RoboDK station: New Station (2).rdk

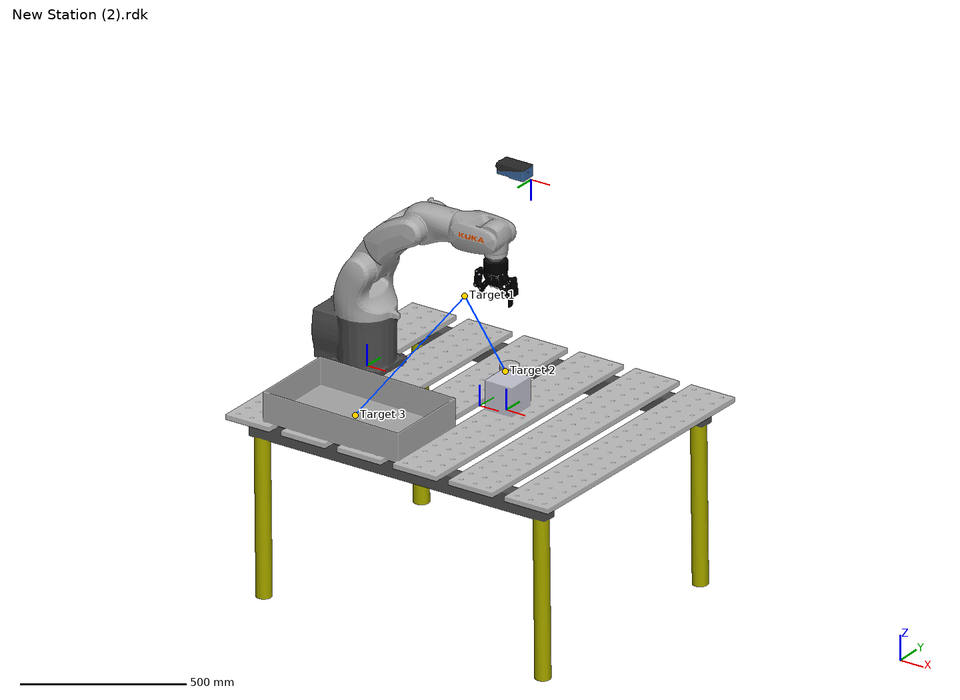
[picture v0: the station drawn from its stored meshes, robots at their saved joint values, targets as dots, program paths as lines]
Station New Station (2). Poses are relative to the parent item; angles as X-Y-Z fixed-axis rotations.
Station parameters (name, value as stored): IO_5, 1, CollisionFreePlanner, KUKA KR 3 R540, CollisionFreePlanner-Rob KUKA KR 3 R540
  - frame KUKA KR 3 R540 Base at (-517.33, 1.06, 0.26) mm, rotated rx -0.44 ry -1.04 rz -0.63 deg
    - robot KUKA KR 3 R540: 6 axes, payload 3 kg, reach 541 mm, repeatability 0.02 mm, weight 26 kg
        modified DH rows (alpha deg, a mm, theta deg, d mm): 0, 0, 0, 345; -90, 20, 0, 0; 0, 260, -90, 0; -90, 20, 0, 260; 90, 0, 0, 0; -90, 0, 180, 75
        joint limits [-170, -170, -110, -175, -120, -350] to [170, 50, 155, 175, 120, 350]; home [0, -90, 90, 0, 0, 0]; saved at [-2.236, -43.368, 43.433, -0.46, 90.207, -1.607]
      - tool Gripper RobotiQ 85 Opened, TCP at (0, -20, 130) mm, size 147.4 x 146.8 x 75 mm
      - tool Gripper RobotiQ 85 Closed, TCP at (0, -20, 130) mm, size 134.4 x 157.6 x 75 mm
    - frame Frame 2 at (440.16, -30.43, -6.02) mm
      - target Target 1 (Cartesian target) at (-55.66, 5.41, 346.75) mm, rotated rx -180 ry 0.75 rz 180 deg; joints [0.676, -64.85, 76.675, 0.003, 78.427, 0.675] of KUKA KR 3 R540
      - target Target 2 (Cartesian target) at (6.97, 122.8, 68.55) mm, rotated rx 180 ry 0.75 rz -180 deg; joints [-14.168, -20.802, 65.869, -0.087, 45.177, -14.106] of KUKA KR 3 R540
      - target Target 3 (Cartesian target) at (-168.25, -408.46, 82.33) mm, rotated rx -180 ry 0.75 rz 180 deg; joints [56.988, -14.801, 48.393, 0.254, 56.546, 56.848] of KUKA KR 3 R540
      - object Table at (0, 0, 0) mm, size 1193.8 x 965.2 x 609.6 mm, geometry from welding_table.sld
    - frame Camera Frame at (617.07, -0.63, 780.12) mm, rotated rx -179.13 ry 0 rz 0 deg
      - object SICK VSPP-5f2113 at (-36.13, -0.26, 0) mm, size 53 x 116 x 38 mm, geometry from Cam2D_SICK_VSPP_5F2113.sld
  - program Prog1 (17 instructions, listed below)
  - frame Frame 3 at (0, -6.9, 0) mm
    - object Box v1 at (-52.65, -189.24, 0) mm, rotated rx 0 ry 0 rz -90.31 deg, size 300 x 500 x 100 mm, geometry from Box v1.stl
  - program Replace objects (1 instructions, listed below)
  - Python program SimulateToolOpen (listed below)
  - Python program SimulateCamera (listed below)
  - object box at (0, 0, 52.21) mm, size 100 x 100 x 100 mm, geometry from box.sld
  - object Part at (-69.82, 109.61, 45.02) mm, size 60 x 60 x 80 mm, geometry from part.sld
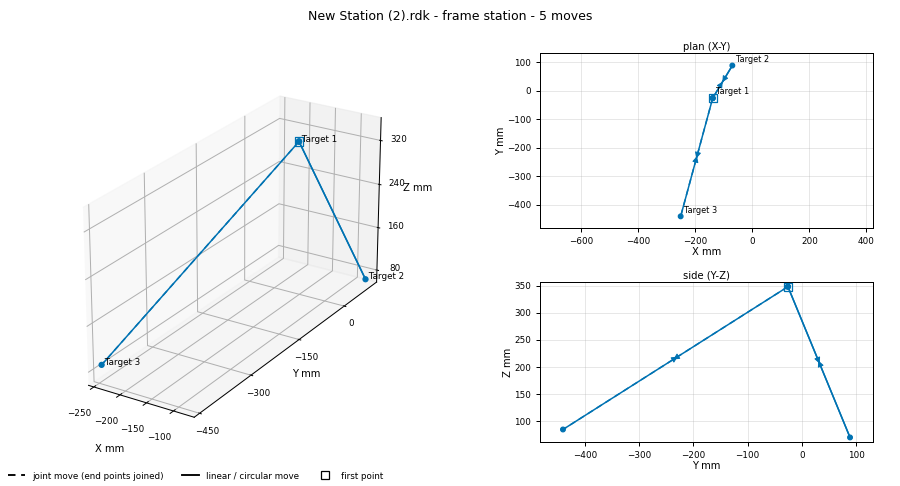
[picture p0: tool path of New Station (2).rdk in frame station, 5 of 5 moves have a stored position in this frame; points joined in program order, loops and branches not executed]

--- program Prog1 (robot KUKA KR 3 R540) ---
  Set speed (100.0 mm/s)
  Set Tool: Gripper RobotiQ 85 Opened at (0, -20, 130) mm
  Call VisibleGripper RobotiQ ...: VisibleGripper RobotiQ 85 Opened_Off
  Set Ref.: Frame 2
  MoveL (Target 1)
  MoveL (Target 2)
  Pause 70 ms
  Attach to Gripper RobotiQ 85 Opened
  Pause 70 ms
  Set Ref.: Frame 3
  MoveL (Target 1)
  MoveJ (Target 3)
  Pause 90 ms
  Detach from Gripper RobotiQ 85 Opened
  Pause 90 ms
  MoveL (Target 1)
  Call Replace objects

--- program Replace objects (robot KUKA KR 3 R540) ---
  Replace objects

--- Python program SimulateToolOpen ---
# Type help("robolink") or help("robodk") for more information
# Press F5 to run the script
# Note: you do not need to keep a copy of this file, your python script is saved with the station
from robolink import *    # API to communicate with RoboDK
from robodk import *      # basic matrix operations
RDK = Robolink()

# This file allows simulating the opening and closing of grippers.
# Two models of the gripper per robot are required: one opened and one closed.
# The opened model of the gripper should have the keyword "Opened"
# The closed model of the gripper should have the keyword "Closed"
# Simply place this file in the station and leave it running to
# make it work

OPENED_KEYWORD = 'Opened'
CLOSED_KEYWORD = 'Closed'
UPDATE_FREQUENCY = 0.01

# Loop forever
print('Starting infinite loop to simulate open/close of tools')
while True:
    # First step: get a list of tool pairs (open, closed) per robot
    Tool_Pairs = []
    # get all the robot names (strings)
    all_robots = RDK.ItemList(ITEM_TYPE_ROBOT, True)
    for i in range(len(all_robots)):
        roboti = RDK.Item(all_robots[i])
        roboti_name = roboti.Name()
        # get the tools of each robot
        roboti_tools = roboti.Childs()
        opened = None
        closed = None
        # store the opened model and closed model of each gripper
        for t in range(len(roboti_tools)):
            tnamei = roboti_tools[t].Name()
            if not isinstance(opened,Item) and tnamei.count(OPENED_KEYWORD) > 0:
                opened = roboti_tools[t]
                print('Using %s from robot %s as gripper opened' % (tnamei, roboti_name))
            elif not isinstance(closed,Item) and tnamei.count(CLOSED_KEYWORD) > 0:
                closed = roboti_tools[t]
                print('Using %s from robot %s as gripper closed' % (tnamei, roboti_name))

            if isinstance(opened, Item) and isinstance(closed, Item):
                # Stop if we have an open state and a closed state per robot
                break;
        Tool_Pairs.append([opened, closed])

    # We may find as many pairs of tools as robots are available in the station
    nTool_Pairs = len(Tool_Pairs)
    while True:
        #try:
            # Iterate through all tool pairs and detect the presence of objects
            for i in range(nTool_Pairs):
                opened = Tool_Pairs[i][0]
                closed = Tool_Pairs[i][1]
                open_valid = isinstance(opened,Item)
                close_valid = isinstance(closed,Item)
                tool_is_open = True

                # Check if the tool holds one or more objects:
                if (open_valid and len(opened.Childs()) > 0) or (close_valid and len(closed.Childs()) > 0):
                    tool_is_open = False

                # Update the visibility of the tools
                if open_valid:
                    opened.setVisible(tool_is_open)
                if close_valid:
                    closed.setVisible(not tool_is_open)

            # Take a pause...
            pause(UPDATE_FREQUENCY)

        #except:
            #print('An item was deleted. Remaking tool list')
            #break

--- Python program SimulateCamera ---
# Type help("robolink") or help("robodk") for more information
# Press F5 to run the script
# Documentation: https://robodk.com/doc/en/RoboDK-API.html
# Reference:     https://robodk.com/doc/en/PythonAPI/index.html
# Note: It is not required to keep a copy of this file, your python script is saved with the station
from robolink import *    # RoboDK API
from robodk import *      # Robot toolbox
RDK = Robolink()

# Notify user:
print('To edit this program:\nright click on the Python program, then, select "Edit Python script"')

# Program example:
item = RDK.Item('base')
if item.Valid():
    print('Item selected: ' + item.Name())
    print('Item posistion: ' + repr(item.Pose()))

print('Items in the station:')
itemlist = RDK.ItemList()
print(itemlist)

raise Exception('Program not edited.')
